FUNCTION TryConvert_WORD_TO_REAL : BOOL
VAR_INPUT
	in : WORD;
	out : REFERENCE TO REAL;
END_VAR

out := WORD_TO_REAL(in);
TryConvert_WORD_TO_REAL := TRUE;

END_FUNCTION

(* stored: Version 1.1.0.1, ProductVersion 3.1.4024.12
   POU TryConvert_WORD_TO_REAL: Id {54a47e00-f377-4e83-9849-c8b42a390f52}, SpecialFunc None *)
